// 40 Visualizations/POPUP/MANUAL/VIS_SENSOR_MANUAL
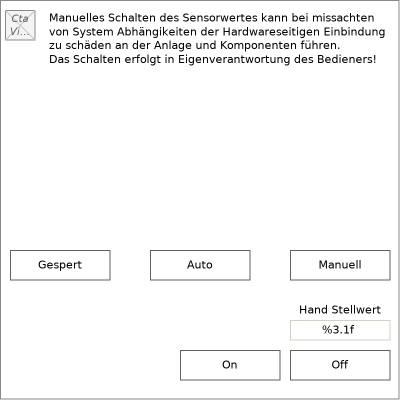
VISUALIZATION VIS_SENSOR_MANUAL  // 400x400
VAR_INPUT
    ITF_SENSORIN    :   ITF_SENSOR;	
END_VAR
    Label (46,10 350x100), "Manuelles Schalten des Sensorwertes kann bei missachten von System Abhängikeiten der Hardwareseitigen Einbindung zu schäden an der Anlage und Komponenten führen. Das Schalten erfolgt in Eigenverantwortung des Bedieners!"
    Textfield (290,320 100x20), "%3.1f", text variable: ITF_SENSORIN.proHandOnY, invisible if: ITF_SENSORIN.proValueInputType = 0 OR ITF_SENSORIN.proValueInputType = 2 OR ITF_SENSORIN.proValueInputType = 4
        OnMouseClick: write the text variable via InputWithLimits, min 0, max 100, title 'Stellwert'
    Image (5,10 30x30), image: CtaVisSymbols.ImagePool.CtaWarning
    Label (290,300 100x20), "Hand Stellwert"
    RoundedRectangle (10,250 100x30), "Gespert", colour toggle: ITF_SENSORIN.proHandOff
        toggle ITF_SENSORIN.proHandOff
    RoundedRectangle (150,250 100x30), "Auto", colour toggle: ITF_SENSORIN.proAuto
        toggle ITF_SENSORIN.proAuto
    RoundedRectangle (290,250 100x30), "Manuell", colour toggle: ITF_SENSORIN.proHandOn
        toggle ITF_SENSORIN.proHandOn
    RoundedRectangle (180,350 100x30), "On", colour toggle: ITF_SENSORIN.proManualTrue, invisible if: ITF_SENSORIN.proValueInputType = 0 OR ITF_SENSORIN.proValueInputType = 1 OR ITF_SENSORIN.proValueInputType = 3
        OnMouseClick: execute { ITF_SENSORIN.proManualTrue := TRUE; }
    RoundedRectangle (290,350 100x30), "Off", colour toggle: ITF_SENSORIN.proManualFalse, invisible if: ITF_SENSORIN.proValueInputType = 0 OR ITF_SENSORIN.proValueInputType = 1 OR ITF_SENSORIN.proValueInputType = 3
        OnMouseClick: execute { ITF_SENSORIN.proManualFalse := TRUE; }
END_VISUALIZATION

// 40 Visualizations/POPUP/OVERVIEW/VIS_SENSOR_OVERVIEW
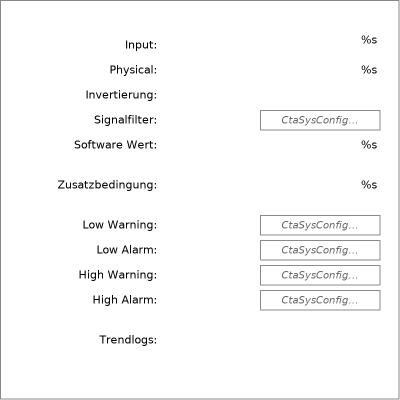
VISUALIZATION VIS_SENSOR_OVERVIEW  // 400x400
VAR_INPUT
    ITF_SENSORIN	:	ITF_SENSOR;
END_VAR
    Frame (0,0 400x400), invisible if: NOT __QUERYINTERFACE(ITF_SENSORIN,ITF_SENSORIN)
        shows VIS_SENSOR_OVERVIEW0(ITF_SENSORIN := ITF_SENSORIN)
END_VISUALIZATION

// 40 Visualizations/POPUP/PARAMETER/SENSOR_ReportManagement/Sensor_HighAlarm_Param
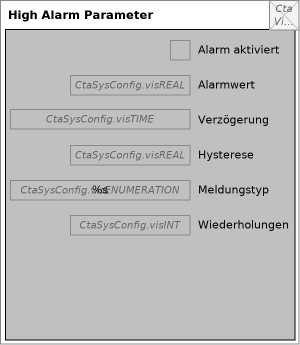
VISUALIZATION Sensor_HighAlarm_Param  // 300x345
VAR_INPUT
	ITF_SENSORIN	:	ITF_SENSOR;
END_VAR
VAR_IN_OUT
    xShow   :   BOOL;
END_VAR
    RoundedRectangle (0,0 299x344)
    RoundedRectangle (5,29 290x311)
    Image (269,0 30x30), image: CtaVisSymbols.ImagePool.close_solo_black
        OnMouseClick: execute { xShow := FALSE; }
    Label (5,0 198x30), "High Alarm Parameter"
    Label (195,40 100x20), "Alarm aktiviert"
    Frame (170,40 20x20)
        shows CtaSysConfig.visBOOL(visfbBOOLIn := ITF_SENSORIN.P_scHighAlram_fbxDoesAlarm)
    Label (195,75 100x20), "Alarmwert"
    Frame (70,75 120x20), invisible if: (ITF_SENSORIN.proValueInputType = enInputType.DigitalInput) OR (ITF_SENSORIN.proValueInputType = enInputType.Digital_ITF_Input)
        shows CtaSysConfig.visREAL(visfbREALIn := ITF_SENSORIN.P_scHighAlarm_fbrValue)
    Label (195,110 100x20), "Verzögerung"
    Frame (10,109 180x20)
        shows CtaSysConfig.visTIME(visfbTIMEIn := ITF_SENSORIN.P_scHighAlarm_fbtDelayTillAlarm)
    Frame (70,145 120x20), invisible if: (ITF_SENSORIN.proValueInputType = enInputType.DigitalInput) OR (ITF_SENSORIN.proValueInputType = enInputType.Digital_ITF_Input)
        shows CtaSysConfig.visREAL(visfbREALIn := ITF_SENSORIN.P_scHighAlarm_fbrHysterese)
    Label (195,145 100x20), "Hysterese"
    Frame (10,180 180x20)
        shows CtaSysConfig.visENUMERATION(visfbENUIn := ITF_SENSORIN.P_scHighAlarm_fbiTypeOfAcknolage)
    Label (195,180 100x20), "Meldungstyp"
    Frame (70,215 120x20), invisible if: NOT (CtaSysConfig.fcGetEnumerationId(ITF_SENSORIN.P_scHighAlarm_fbiTypeOfAcknolage) = 2)
        shows CtaSysConfig.visINT(visfbINTIn := ITF_SENSORIN.P_scHighAlarm_fbiRetryTillLock)
    Label (195,215 100x20), "Wiederholungen"
    Textfield (30,180 140x20), "%s", text list: 'CtaAppReport.txtLibAp99_2enTypeOfAck', text index: CtaSysConfig.fcGetEnumerationId(ITF_SENSORIN.P_scHighAlarm_fbiTypeOfAcknolage)
END_VISUALIZATION

// 40 Visualizations/ICON/SENSOR_FLAT/SENSOR_FLAT_TXT_LEFT/BELOW/VIS_SENSOR_FLAT_LEFT_BELOW
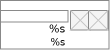
VISUALIZATION VIS_SENSOR_FLAT_LEFT_BELOW  // 110x50
VAR_INPUT
    ITF_SENSOR_IN   :   ITF_SENSOR;	
END_VAR
VAR_INPUT CONSTANT	
	stExklParameter	:	STRING [40] := ' ';	
END_VAR
VAR CONSTANT
	uiIconNr		: UINT := 1;
END_VAR
    Frame (0,0 110x50), invisible if: NOT fcCheckQuerryAndIconReturn(_ITF_IN := ITF_SENSOR_IN, _uiIconNr_IN := uiIconNr)
        shows VIS_SENSOR_FLAT_LeftBelowCheckQuerry(ITF_SENSOR_IN := ITF_SENSOR_IN, stExklParameter := stExklParameter)
END_VISUALIZATION

// 40 Visualizations/POPUP/PARAMETER/SENSOR_ReportManagement/Sensor_HighWarning_Param
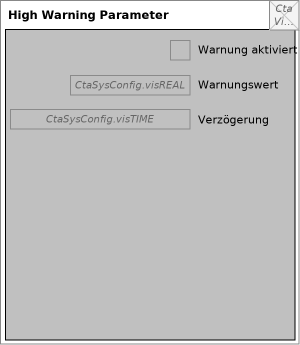
VISUALIZATION Sensor_HighWarning_Param  // 300x345
VAR_INPUT
	ITF_SENSORIN	:	ITF_SENSOR;
END_VAR
VAR_IN_OUT
    xShow   :   BOOL;
END_VAR
    RoundedRectangle (0,0 299x344)
    RoundedRectangle (5,29 290x311)
    Image (269,0 30x30), image: CtaVisSymbols.ImagePool.close_solo_black
        OnMouseClick: execute { xShow := FALSE; }
    Label (5,0 198x30), "High Warning Parameter"
    Label (195,40 100x20), "Warnung aktiviert"
    Frame (170,40 20x20)
        shows CtaSysConfig.visBOOL(visfbBOOLIn := ITF_SENSORIN.P_scHighWarning_fbxDoesWarning)
    Label (195,75 100x20), "Warnungswert"
    Frame (70,75 120x20), invisible if: (ITF_SENSORIN.proValueInputType = enInputType.DigitalInput) OR (ITF_SENSORIN.proValueInputType = enInputType.Digital_ITF_Input)
        shows CtaSysConfig.visREAL(visfbREALIn := ITF_SENSORIN.P_scHighWarning_fbrValue)
    Label (195,110 100x20), "Verzögerung"
    Frame (10,109 180x20)
        shows CtaSysConfig.visTIME(visfbTIMEIn := ITF_SENSORIN.P_scHighWarning_fbtDelayTillWarning)
END_VISUALIZATION

// 40 Visualizations/ICON/SENSOR_FLAT/SENSOR_FLAT_TXT_LEFT/BELOW/VIS_SENSOR_FLAT_LeftBelowCheckIsEnabled
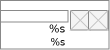
VISUALIZATION VIS_SENSOR_FLAT_LeftBelowCheckIsEnabled  // 110x50
VAR_INPUT
    ITF_SENSOR_IN   :   ITF_SENSOR;
	stExklParameter	:	STRING [40];	
END_VAR
    Frame (70,10 38x20), invisible if: NOT ITF_SENSOR_IN.proIsEnabled
        shows SensorFlat(ITF_SENSORIN := ITF_SENSOR_IN)
    Frame (0,10 68x40), invisible if: NOT ITF_SENSOR_IN.proIsEnabled
        shows ValueDwnUp(ITF_SENSORIN := ITF_SENSOR_IN, uiTextAusrichtung := 6)
    Rectangle (0,0 110x50)
        OnMouseClick:  Dialog=POPUP_SENSOR, Parameters={stExklParameter: stExklParameter, ITF_SENSORIN: ITF_SENSOR_IN, uiPopUpGruppe: 0}, OpenCentered=True
END_VISUALIZATION

// 40 Visualizations/POPUP/REPORTS/VIS_SENSOR_REPORTS
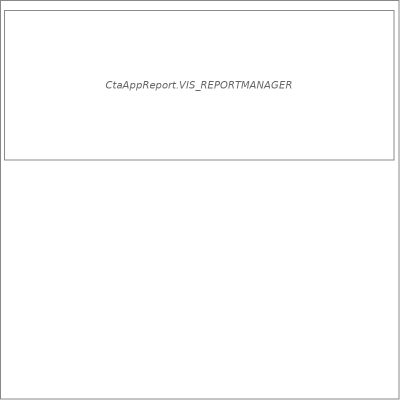
VISUALIZATION VIS_SENSOR_REPORTS  // 400x400
VAR_INPUT
    ITF_SENSORIN    :   ITF_SENSOR;	
END_VAR
    Frame (4,10 390x150)
        shows CtaAppReport.VIS_REPORTMANAGER(ITF_REPORTMANAGER := ITF_SENSORIN.proITF_REPORTMANAGER)
END_VISUALIZATION

// 40 Visualizations/POPUP/PARAMETER/SENSOR_ParameterBase/VIS_SENSOR_PARAMETER_BASE0
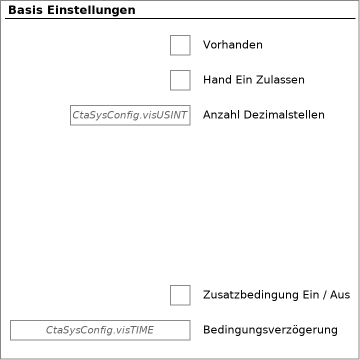
VISUALIZATION VIS_SENSOR_PARAMETER_BASE0  // 360x360
VAR_INPUT
    ITF_SENSORIN	:  ITF_SENSOR;
END_VAR
    Label (5,0 350x20), "Basis Einstellungen"
    Line (5,18) (355,18)
    Label (200,35 150x20), "Vorhanden"
    Label (200,70 150x20), "Hand Ein Zulassen"
    Frame (170,35 20x20)
        shows CtaSysConfig.visBOOL(visfbBOOLIn := ITF_SENSORIN.P_scBase_fbxEnable)
    Frame (170,70 20x20)
        shows CtaSysConfig.visBOOL(visfbBOOLIn := ITF_SENSORIN.P_scManual_fbxAllowManualOn)
    Frame (170,285 20x20)
        shows CtaSysConfig.visBOOL(visfbBOOLIn := ITF_SENSORIN.P_scAlCondition_fbxEnable)
    Label (200,285 150x20), "Zusatzbedingung Ein / Aus"
    Frame (10,320 180x20)
        shows CtaSysConfig.visTIME(visfbTIMEIn := ITF_SENSORIN.P_scAlCondition_fbtDelayTillCondition)
    Label (200,320 150x20), "Bedingungsverzögerung"
    Frame (70,105 120x20), invisible if: NOT (ITF_SENSORIN.proValueInputType = enInputType.AnalogInput or ITF_SENSORIN.proValueInputType = enInputType.Analog_ITF_Input)
        shows CtaSysConfig.visUSINT(visfbUSINTIn := ITF_SENSORIN.P_scVisu_fbusiDezimalPos)
    Label (200,105 150x20), "Anzahl Dezimalstellen", invisible if: NOT (ITF_SENSORIN.proValueInputType = enInputType.AnalogInput or ITF_SENSORIN.proValueInputType = enInputType.Analog_ITF_Input)
END_VISUALIZATION

// 40 Visualizations/POPUP/PARAMETER/SENSOR_ParameterBase/VIS_SENSOR_PARAMETER_BASE
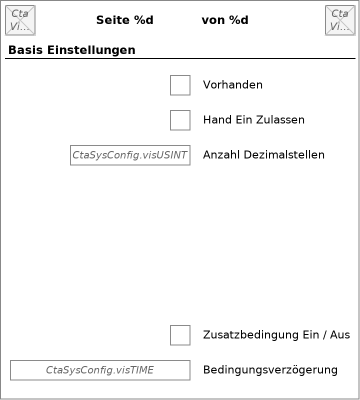
VISUALIZATION VIS_SENSOR_PARAMETER_BASE  // 360x400
VAR_INPUT
    ITF_SENSORIN 	: 	ITF_SENSOR;
END_VAR
VAR
    uiPage  :   UINT;
    uiMin   :   UINT    := 0;
    uiMax   :   UINT    := 0;
END_VAR
    Image (5,5 30x30), invisible if: uiPage = uiMin, image: CtaVisSymbols.ImagePool.arrow-left_square
        OnMouseClick: execute {
            uiPage := uiPage - 1;
            IF uiPage <= uiMin THEN
                uiPage := uiMin;
            END_IF;
        }
    Image (325,5 30x30), invisible if: uiPage = uiMax, image: CtaVisSymbols.ImagePool.arrow-right_square
        OnMouseClick: execute {
            uiPage := uiPage + 1;
            IF uiPage >= uiMax THEN
                uiPage := uiMax;
            END_IF;
        }
    Frame (0,40 360x360), frame switch variable: uiPage
        shows VIS_SENSOR_PARAMETER_BASE0(ITF_SENSORIN := ITF_SENSORIN)
        shows AT_ParameterIO1(ITF_Parameter := ITF_Parameter)
        pReferences[0]: ITF_Parameter=ITF_Parameter
    Textfield (175,5 100x30), "von %d", text variable: uiMax
    Textfield (75,5 100x30), "Seite %d", text variable: uiPage
END_VISUALIZATION

// 40 Visualizations/ICON/SENSOR_FLAT/SENSOR_FLAT_TXT_RIGHT/ABOVE/VIS_SENSOR_FLAT_RIGHT_ABOVE
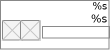
VISUALIZATION VIS_SENSOR_FLAT_RIGHT_ABOVE  // 110x50
VAR_INPUT
    ITF_SENSOR_IN   :   ITF_SENSOR;	
END_VAR
VAR_INPUT CONSTANT	
	stExklParameter	:	STRING [40] := ' ';	
END_VAR
VAR CONSTANT
	uiIconNr		:	UINT := 2;
END_VAR
    Frame (0,0 110x50), invisible if: NOT fcCheckQuerryAndIconReturn(_ITF_IN := ITF_SENSOR_IN, _uiIconNr_IN := uiIconNr)
        shows VIS_SENSOR_FLAT_RigthAboveCheckQuerry(ITF_SENSOR_IN := ITF_SENSOR_IN, stExklParameter := stExklParameter)
END_VISUALIZATION

// 40 Visualizations/ICON/SENSOR_FLAT/SENSOR_FLAT_TXT_LEFT/BELOW/VIS_SENSOR_FLAT_LeftBelowCheckQuerry
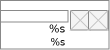
VISUALIZATION VIS_SENSOR_FLAT_LeftBelowCheckQuerry  // 110x50
VAR_INPUT
    ITF_SENSOR_IN   :   ITF_SENSOR;
	stExklParameter	:	STRING [40];	
END_VAR
    Frame (0,0 110x50)
        shows VIS_SENSOR_FLAT_LeftBelowCheckIsEnabled(ITF_SENSOR_IN := ITF_SENSOR_IN, stExklParameter := stExklParameter)
END_VISUALIZATION

// 40 Visualizations/POPUP/PARAMETER/SENSOR_ReportManagement/VIS_SENSOR_PARAMETER_REPORTMNG
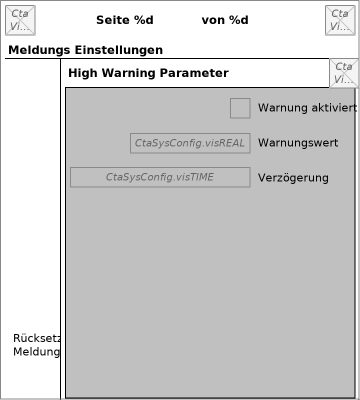
VISUALIZATION VIS_SENSOR_PARAMETER_REPORTMNG  // 360x400
VAR_INPUT
   	ITF_SENSORIN	:	ITF_SENSOR;
END_VAR
VAR
    uiPage  :   UINT;
    uiMin   :   UINT    := 0;
    uiMax   :   UINT    := 0;
END_VAR
    Image (5,5 30x30), invisible if: uiPage = uiMin, image: CtaVisSymbols.ImagePool.arrow-left_square
        OnMouseClick: execute {
            uiPage := uiPage - 1;
            IF uiPage <= uiMin THEN
                uiPage := uiMin;
            END_IF;
        }
    Image (325,5 30x30), invisible if: uiPage = uiMax, image: CtaVisSymbols.ImagePool.arrow-right_square
        OnMouseClick: execute {
            uiPage := uiPage + 1;
            IF uiPage >= uiMax THEN
                uiPage := uiMax;
            END_IF;
        }
    Frame (0,40 360x360), frame switch variable: uiPage
        shows VIS_SENSOR_PARAMETER_REPORTMNG_1(ITF_SENSORIN := ITF_SENSORIN)
        shows AT_ParameterIO1(ITF_Parameter := ITF_Parameter)
    Textfield (175,5 100x30), "von %d", text variable: uiMax
    Textfield (75,5 100x30), "Seite %d", text variable: uiPage
END_VISUALIZATION

// 40 Visualizations/POPUP/PARAMETER/SENSOR_ReportManagement/VIS_SENSOR_PARAMETER_REPORTMNG_1
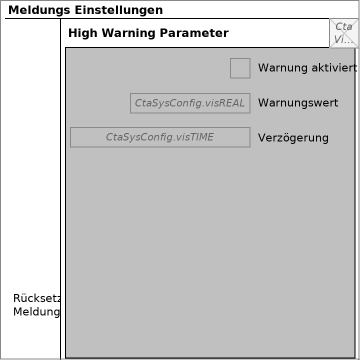
VISUALIZATION VIS_SENSOR_PARAMETER_REPORTMNG_1  // 360x360
VAR_INPUT
   	ITF_SENSORIN	:	ITF_SENSOR;
END_VAR
VAR
	xShowLoWarning	:	BOOL;
	xShowLoAlarm	:	BOOL;
	xShowHiWarning	:	BOOL;
	xShowHiAlarm	:	BOOL;
END_VAR
    Label (5,0 350x20), "Meldungs Einstellungen"
    Line (5,18) (355,18)
    Label (200,35 150x20), "Low warning"
    Label (200,80 150x20), "Low alarm"
    Label (200,125 150x20), "High warning"
    Label (200,170 150x20), "High alarm"
    Image (300,30 32x32), image: CtaVisSymbols. ImagePool.CtaInfo
        OnMouseClick: execute {
            xShowLoWarning	:=	TRUE;
            xShowLoAlarm	:=	FALSE;
            xShowHiWarning	:=	FALSE;
            xShowHiAlarm	:=	FALSE;
        }
    Image (300,75 32x32), image: CtaVisSymbols.ImagePool.CtaInfo
        OnMouseClick: execute {
            xShowLoWarning	:=	FALSE;
            xShowLoAlarm	:=	TRUE;
            xShowHiWarning	:=	FALSE;
            xShowHiAlarm	:=	FALSE;
        }
    Image (300,120 32x32), image: CtaVisSymbols.ImagePool.CtaInfo
        OnMouseClick: execute {
            xShowLoWarning	:=	FALSE;
            xShowLoAlarm	:=	FALSE;
            xShowHiWarning	:=	TRUE;
            xShowHiAlarm	:=	FALSE;
        }
    Image (300,165 32x32), image: CtaVisSymbols.ImagePool.CtaInfo
        OnMouseClick: execute {
            xShowLoWarning	:=	FALSE;
            xShowLoAlarm	:=	FALSE;
            xShowHiWarning	:=	FALSE;
            xShowHiAlarm	:=	TRUE;
        }
    Frame (170,230 20x20)
        shows CtaSysConfig.visBOOL(visfbBOOLIn := ITF_SENSORIN.P_scAnalogAlarm_fbxEnableOverflowAl)
    Label (200,230 160x20), "Alarm Überlauf aktiviert"
    Label (200,265 160x20), "Alarm Unterlauf aktiviert"
    Frame (170,265 20x20)
        shows CtaSysConfig.visBOOL(visfbBOOLIn := ITF_SENSORIN.P_scAnalogAlarm_fbxEnableUnderflowAl)
    Frame (170,300 180x20)
        shows CtaSysConfig.visTIME(visfbTIMEIn := ITF_SENSORIN.P_scAlarmReset_fbtDealyTillReset)
    Label (10,285 160x40), "Rücksetzung des Retry - N Meldungszählers nach:"
    Frame (60,18 300x345), invisible if: NOT xShowHiAlarm
        shows Sensor_HighAlarm_Param(ITF_SENSORIN := ITF_SENSORIN, xShow := xShowHiAlarm)
    Frame (60,18 300x345), invisible if: NOT xShowLoWarning
        shows Sensor_LowWarning_Param(ITF_SENSORIN := ITF_SENSORIN, xShow := xShowLoWarning)
    Frame (60,18 300x345), invisible if: NOT xShowLoAlarm
        shows Sensor_LowAlarm_Param(ITF_SENSORIN := ITF_SENSORIN, xShow := xShowLoAlarm)
    Frame (60,18 300x345), invisible if: NOT xShowHiWarning
        shows Sensor_HighWarning_Param(ITF_SENSORIN := ITF_SENSORIN, xShow := xShowHiWarning)
END_VISUALIZATION

// 40 Visualizations/POPUP/PARAMETER/SENSOR_Filter/VIS_SENSOR_PARAMETER_FILTER
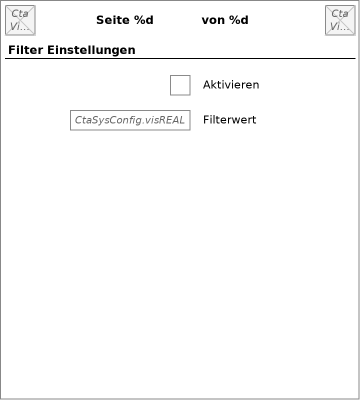
VISUALIZATION VIS_SENSOR_PARAMETER_FILTER  // 360x400
VAR_INPUT
  	ITF_SENSORIN	:	ITF_SENSOR;
END_VAR
VAR
    uiPage  :   UINT;
    uiMin   :   UINT    := 0;
    uiMax   :   UINT    := 0;
END_VAR
    Image (5,5 30x30), invisible if: uiPage = uiMin, image: CtaVisSymbols.ImagePool.arrow-left_square
        OnMouseClick: execute {
            uiPage := uiPage - 1;
            IF uiPage <= uiMin THEN
                uiPage := uiMin;
            END_IF;
        }
    Image (325,5 30x30), invisible if: uiPage = uiMax, image: CtaVisSymbols.ImagePool.arrow-right_square
        OnMouseClick: execute {
            uiPage := uiPage + 1;
            IF uiPage >= uiMax THEN
                uiPage := uiMax;
            END_IF;
        }
    Frame (0,40 360x360), frame switch variable: uiPage
        shows VIS_SENSOR_PARAMETER_FILTER_1(ITF_SENSORIN := ITF_SENSORIN)
        shows AT_ParameterIO1(ITF_Parameter := ITF_Parameter)
    Textfield (175,5 100x30), "von %d", text variable: uiMax
    Textfield (75,5 100x30), "Seite %d", text variable: uiPage
END_VISUALIZATION

// 40 Visualizations/POPUP/PARAMETER/SENSOR_Filter/VIS_SENSOR_PARAMETER_FILTER_1
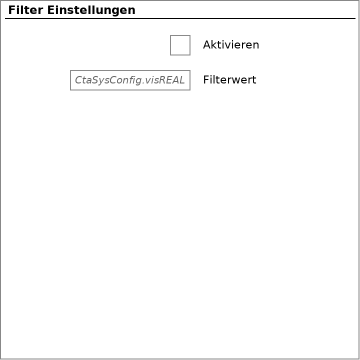
VISUALIZATION VIS_SENSOR_PARAMETER_FILTER_1  // 360x360
VAR_INPUT
   	ITF_SENSORIN	:	ITF_SENSOR;
END_VAR
    Label (5,0 350x20), "Filter Einstellungen"
    Line (5,18) (355,18)
    Frame (170,35 20x20)
        shows CtaSysConfig.visBOOL(visfbBOOLIn := ITF_SENSORIN.P_scFilter_fbxEnabled)
    Label (200,35 150x20), "Aktivieren"
    Frame (70,70 120x20)
        shows CtaSysConfig.visREAL(visfbREALIn := ITF_SENSORIN.P_scFilter_fbrValue)
    Label (200,70 150x20), "Filterwert"
END_VISUALIZATION

// 40 Visualizations/POPUP/PARAMETER/SENSOR_InfluxDb/VIS_SENSOR_PARAMETER_TRENDLOG
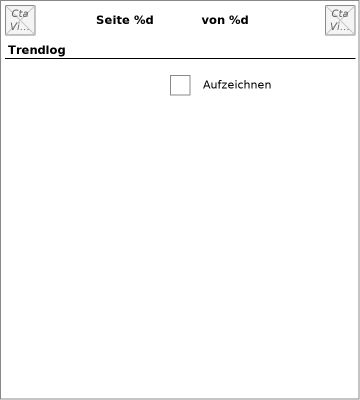
VISUALIZATION VIS_SENSOR_PARAMETER_TRENDLOG  // 360x400
VAR_INPUT
   	ITF_SENSORIN	:	ITF_SENSOR;
END_VAR
VAR
    uiPage  :   UINT;
    uiMin   :   UINT    := 0;
    uiMax   :   UINT    := 0;
END_VAR
    Image (5,5 30x30), invisible if: uiPage = uiMin, image: CtaVisSymbols.ImagePool.arrow-left_square
        OnMouseClick: execute {
            uiPage := uiPage - 1;
            IF uiPage <= uiMin THEN
                uiPage := uiMin;
            END_IF;
        }
    Image (325,5 30x30), invisible if: uiPage = uiMax, image: CtaVisSymbols.ImagePool.arrow-right_square
        OnMouseClick: execute {
            uiPage := uiPage + 1;
            IF uiPage >= uiMax THEN
                uiPage := uiMax;
            END_IF;
        }
    Frame (0,40 360x360), frame switch variable: uiPage
        shows VIS_SENSOR_PARAMETER_TRENDLOG0(ITF_SENSORIN := ITF_SENSORIN)
        shows AT_ParameterIO1(ITF_Parameter := ITF_Parameter)
        pReferences[0]: ITF_Parameter=ITF_Parameter
    Textfield (75,5 100x30), "Seite %d", text variable: uiPage
    Textfield (175,5 100x30), "von %d", text variable: uiMax
END_VISUALIZATION

// 40 Visualizations/POPUP/PARAMETER/SENSOR_InfluxDb/VIS_SENSOR_PARAMETER_TRENDLOG0
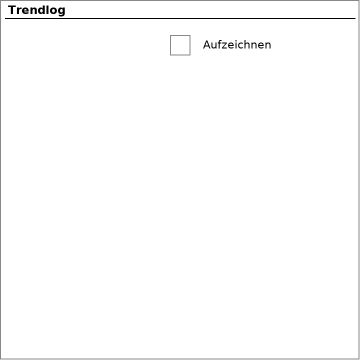
VISUALIZATION VIS_SENSOR_PARAMETER_TRENDLOG0  // 360x360
VAR_INPUT
    ITF_SENSORIN	:	ITF_SENSOR;
END_VAR
    Frame (170,35 20x20)
        shows CtaSysConfig.visBOOL(visfbBOOLIn := ITF_SENSORIN.P_scInfluxDb_fbxEnable)
    Label (200,35 150x20), "Aufzeichnen"
    Label (5,0 350x20), "Trendlog"
    Line (5,18) (355,18)
END_VISUALIZATION

// 40 Visualizations/POPUP/PARAMETER/SENSOR_ReportManagement/Sensor_LowWarning_Param
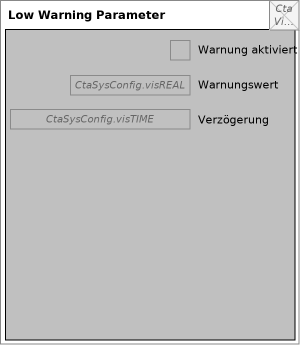
VISUALIZATION Sensor_LowWarning_Param  // 300x345
VAR_INPUT
	ITF_SENSORIN	:	ITF_SENSOR;
END_VAR
VAR_IN_OUT
    xShow   :   BOOL;
END_VAR
    RoundedRectangle (0,0 299x344)
    RoundedRectangle (5,29 290x311)
    Image (269,0 30x30), image: CtaVisSymbols.ImagePool.close_solo_black
        OnMouseClick: execute { xShow := FALSE; }
    Label (5,0 198x30), "Low Warning Parameter"
    Label (195,40 100x20), "Warnung aktiviert"
    Frame (170,40 20x20)
        shows CtaSysConfig.visBOOL(visfbBOOLIn := ITF_SENSORIN.P_scLoWarning_fbxDoesWarning)
    Label (195,75 100x20), "Warnungswert"
    Frame (70,75 120x20), invisible if: (ITF_SENSORIN.proValueInputType = enInputType.DigitalInput) OR (ITF_SENSORIN.proValueInputType = enInputType.Digital_ITF_Input)
        shows CtaSysConfig.visREAL(visfbREALIn := ITF_SENSORIN.P_scLoWarning_fbrValue)
    Label (195,110 100x20), "Verzögerung"
    Frame (10,109 180x20)
        shows CtaSysConfig.visTIME(visfbTIMEIn := ITF_SENSORIN.P_scLoWarning_fbtDelayTillWarning)
END_VISUALIZATION

// 40 Visualizations/ICON/SENSOR_FLAT/SENSOR_FLAT_TXT_RIGHT/ABOVE/VIS_SENSOR_FLAT_RigthAboveCheckQuerry
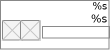
VISUALIZATION VIS_SENSOR_FLAT_RigthAboveCheckQuerry  // 110x50
VAR_INPUT
    ITF_SENSOR_IN   :   ITF_SENSOR;
	stExklParameter	:	STRING [40];
END_VAR
    Frame (0,0 110x50)
        shows VIS_SENSOR_FLAT_RigthAboveCheckIsEnabled(ITF_SENSOR_IN := ITF_SENSOR_IN, stExklParameter := stExklParameter)
END_VISUALIZATION

// 40 Visualizations/ICON/SENSOR_ROUND/SENSOR_ROUNF_TXT_LEFT/ABOVE/VIS_SENSOR_ROUND_LEFT_ABOVE
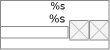
VISUALIZATION VIS_SENSOR_ROUND_LEFT_ABOVE  // 110x50
VAR_INPUT
    ITF_SENSOR_IN   :   ITF_SENSOR;	
END_VAR
VAR_INPUT CONSTANT	
	stExklParameter	:	STRING [40] := ' ';	
END_VAR
VAR CONSTANT
	uiIconnr		:	UINT := 6;
END_VAR
    Frame (0,0 110x50), invisible if: NOT fcCheckQuerryAndIconReturn(_ITF_IN := ITF_SENSOR_IN, _uiIconNr_IN := uiIconNr)
        shows VIS_SENSOR_ROUND_LeftAboveCheckQuerry(ITF_SENSOR_IN := ITF_SENSOR_IN, stExklParameter := stExklParameter)
END_VISUALIZATION

// 40 Visualizations/ICON/SENSOR_ROUND/SENSOR_ROUNF_TXT_LEFT/ABOVE/VIS_SENSOR_ROUND_LeftAboveCheckIsEnabled
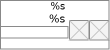
VISUALIZATION VIS_SENSOR_ROUND_LeftAboveCheckIsEnabled  // 110x50
VAR_INPUT
    ITF_SENSOR_IN   :   ITF_SENSOR;
	stExklParameter	:	STRING [40];	
END_VAR
    Frame (69,20 40x20), invisible if: NOT ITF_SENSOR_IN.proIsEnabled
        shows SensorRound(ITF_SENSORIN := ITF_SENSOR_IN)
    Frame (0,0 68x40), invisible if: NOT ITF_SENSOR_IN.proIsEnabled
        shows ValueUpDwn(ITF_SENSORIN := ITF_SENSOR_IN, uiTextAusrichtung := 6)
    Rectangle (0,0 110x50)
        OnMouseClick:  Dialog=POPUP_SENSOR, Parameters={stExklParameter: stExklParameter, ITF_SENSORIN: ITF_SENSOR_IN, uiPopUpGruppe: 0}, OpenCentered=True
END_VISUALIZATION

// 40 Visualizations/ICON/SENSOR_ROUND/SENSOR_ROUNF_TXT_LEFT/ABOVE/VIS_SENSOR_ROUND_LeftAboveCheckQuerry
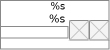
VISUALIZATION VIS_SENSOR_ROUND_LeftAboveCheckQuerry  // 110x50
VAR_INPUT
    ITF_SENSOR_IN   :   ITF_SENSOR;
	stExklParameter	:	STRING [40];	
END_VAR
    Frame (0,0 110x50)
        shows VIS_SENSOR_ROUND_LeftAboveCheckIsEnabled(ITF_SENSOR_IN := ITF_SENSOR_IN, stExklParameter := stExklParameter)
END_VISUALIZATION

// 40 Visualizations/ICON/SENSOR_ROUND/SENSOR_ROUND_TXT_RIGHT/ABOVE/VIS_SENSOR_ROUND_RIGHT_ABOVE
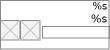
VISUALIZATION VIS_SENSOR_ROUND_RIGHT_ABOVE  // 110x50
VAR_INPUT
    ITF_SENSOR_IN   :   ITF_SENSOR;	
END_VAR
VAR_INPUT CONSTANT	
	stExklParameter	:	STRING [40] := ' ';	
END_VAR
VAR CONSTANT
	uiIconNr		:	UINT := 4;
END_VAR
    Frame (0,0 110x50), invisible if: NOT fcCheckQuerryAndIconReturn(_ITF_IN := ITF_SENSOR_IN, _uiIconNr_IN := uiIconNr)
        shows VIS_SENSOR_ROUND_RightAboveCheckQuerry(ITF_SENSOR_IN := ITF_SENSOR_IN, stExklParameter := stExklParameter)
END_VISUALIZATION

// 40 Visualizations/ICON/SENSOR_ROUND/SENSOR_ROUND_TXT_RIGHT/ABOVE/VIS_SENSOR_ROUND_RightAboveCheckIsEnabled
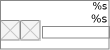
VISUALIZATION VIS_SENSOR_ROUND_RightAboveCheckIsEnabled  // 110x50
VAR_INPUT
    ITF_SENSOR_IN   :   ITF_SENSOR;
	stExklParameter	:	STRING [40];	
END_VAR
    Frame (0,20 40x20), invisible if: NOT ITF_SENSOR_IN.proIsEnabled
        shows SensorRound(ITF_SENSORIN := ITF_SENSOR_IN)
    Frame (42,0 68x40), invisible if: NOT ITF_SENSOR_IN.proIsEnabled
        shows ValueUpDwn(ITF_SENSORIN := ITF_SENSOR_IN, uiTextAusrichtung := 4)
    Rectangle (0,0 110x50)
        OnMouseClick:  Dialog=POPUP_SENSOR, Parameters={stExklParameter: stExklParameter, ITF_SENSORIN: ITF_SENSOR_IN, uiPopUpGruppe: 0}, OpenCentered=True
END_VISUALIZATION

// 40 Visualizations/ICON/SENSOR_ROUND/SENSOR_ROUND_TXT_RIGHT/ABOVE/VIS_SENSOR_ROUND_RightAboveCheckQuerry
